FUNCTION_BLOCK HMIHandler_t
VAR_INPUT
	systemStatus : POINTER TO systemStatus_t;
END_VAR
VAR_OUTPUT
END_VAR
VAR
	_PLCStatusDisplayErrorBlinker : FB_BA_Blink;
END_VAR

METHOD PRIVATE statusDisplayMachine : BOOL
VAR_INPUT
END_VAR
_PLCStatusDisplayErrorBlinker.bEn := TRUE;
_PLCStatusDisplayErrorBlinker.udiTiOff := 500; // 500 ms
_PLCStatusDisplayErrorBlinker.udiTiOn := 500;  // 500 ms
_PLCStatusDisplayErrorBlinker();


CASE systemStatus^ OF
	systemStatus_t.RUNNING:
		HMIInterface.HMIStartStatusLamp := TRUE;
		HMIInterface.HMIStopStatusLamp := FALSE;
		HMIInterface.HMIErrorStatusLamp := FALSE;
		
	systemStatus_t.STOPPED:
		HMIInterface.HMIStartStatusLamp := FALSE;
		HMIInterface.HMIStopStatusLamp := TRUE;
		HMIInterface.HMIErrorStatusLamp := FALSE;

	systemStatus_t.ERROR:	
		HMIInterface.HMIStartStatusLamp := FALSE;
		HMIInterface.HMIStopStatusLamp := FALSE;
		HMIInterface.HMIErrorStatusLamp := _PLCStatusDisplayErrorBlinker.bQ;

END_CASE
END_METHOD

// call this methode every cycle
METHOD update : BOOL
VAR_INPUT
END_VAR
this^.statusDisplayMachine();
END_METHOD

END_FUNCTION_BLOCK

(* stored: Version 1.1.0.1
   POU HMIHandler_t: Id {ceb94381-ed90-43c9-925f-fa3cce5edc0c}, SpecialFunc None
   Method statusDisplayMachine: Id {a22eb489-d856-41a0-81b8-cf1c1e28babf}
   Method update: Id {c2ec0e7d-b831-4ce3-bede-a7d7d46ea402} *)
